FUNCTION_BLOCK FB_HomeNC_Test EXTENDS FB_TestSuite
VAR
    fbAxisRef : ARRAY [1..8] OF AXIS_REF;
    fbLimSwStatus : ARRAY [1..8] OF FB_LimSwStatus_TestDouble;
    //fbMotionLogger : FB_MotionLogger;
    fbMotionLogger : ARRAY [1..8] OF FB_MotionLogger;
    fbPower : ARRAY [1..8] OF FB_PowerNC[	(AxisRef := fbAxisRef[1]),
                                            (AxisRef := fbAxisRef[2]),
                                            (AxisRef := fbAxisRef[3]),
                                            (AxisRef := fbAxisRef[4]),
                                            (AxisRef := fbAxisRef[5]),
                                            (AxisRef := fbAxisRef[6]),
                                            (AxisRef := fbAxisRef[7]),
                                            (AxisRef := fbAxisRef[8])
                                            ];
END_VAR

GivenHomeCmdNoneThenHomeDoneIsTrue_Test1();
GivenHomeCmdAbsoluteSetThenThenAndHomeDoneAndPositionSetToUserDefineOffset_Test2();
GivenHomeCmdLowLimitModeAndABackwardSwPulseThenHomeDoneAndPositionSetToUserDefineOffset_Test3();
GivenHomeCmdSetToHighLimitAndHighLimitPulseThenHomeDoneAndPositionSetToUserDefineOffset_Test4();
GivenHomeCmdSetToHomeViaHighLimitAndHomeHighLimitPulseThenHomeDoneAndPositionSetToUserDefineOffset_Test5();
GivenHomeCmdSetToHomeViaLowLimitAndHomeLowLimitPulseThenHomeDoneAndPositionSetToUserDefineOffset_Test6();
GivenHomeCmdSetToHomeViaLowLimitAndBackwardLimitPulsebeforeHomeLowLimitIdexPulseThenHomeDoneAndPositionSetToUserDefineOffset_Test7();
GivenHomeCmdSetToHomeViaHighLimitAndForwardLimitPulsebeforeHomeHighLimitIdexPulseThenHomeDoneAndPositionSetToUserDefineOffset_Test8();

METHOD PRIVATE GivenHomeCmdAbsoluteSetThenThenAndHomeDoneAndPositionSetToUserDefineOffset_Test2
VAR_INST
    fbHome : FB_HomeNC(AxisRef:=fbAxisRef[2], iLimSwStatus:=fbLimSwStatus[2],iMotionLogger:=fbMotionLogger[2]):=(Mode:=E_EpicsHomeCmd.ABSOLUTE_SET);
    fbTestTimer: TON := (IN:=TRUE, PT:=T#8S);

    nTestStep : INT;
    fExpectedPosition : LREAL := 20.0;
    fActPosition : LREAL;
    bCalibrated : BOOL;
END_VAR
TEST(__POUNAME());

fbLimSwStatus[2]();
fbMotionLogger[2]();
// This methd must be called cyclicly
fbPower[2].Power(	Enable:=TRUE,
                     Enable_Positive:=fbLimSwStatus[2].LimForward,
                       Enable_Negative:=fbLimSwStatus[2].LimBackward,
                       Override:=100.0
                );

CASE nTestStep OF
    0:
        IF fbPower[2].PowerIsEnabled THEN
            fbHome.Home(Position:=20.0,BufferMode:=MC_BufferMode.MC_Aborting);
            nTestStep := nTestStep + 1;
        END_IF
    1:
        IF fbHome.Done THEN
            nTestStep := nTestStep + 1;
        END_IF
    2:
     //
END_CASE
fbAxisRef[2].ReadStatus();
fbHome();
fbTestTimer(IN := TRUE);

IF nTestStep = 2 THEN
bCalibrated := fbHome.Done;
AssertEquals_BOOL(Expected:=fbAxisRef[2].Status.Homed, Actual:=bCalibrated, Message := 'Axis not calibrated #1');

AssertEquals_LREAL ( Delta:=0.001, Expected:=fExpectedPosition, Actual:=fbAxisRef[2].NcToPlc.ActPos, Message:='Position is not the expected #2');
TEST_FINISHED();
ELSIF fbTestTimer.Q THEN
    AssertTrue(
        Condition := FALSE,
        Message := CONCAT('Timed out at step: ', TO_STRING(nTestStep))
    );
    TEST_FINISHED();
END_IF
END_METHOD

METHOD PRIVATE GivenHomeCmdLowLimitModeAndABackwardSwPulseThenHomeDoneAndPositionSetToUserDefineOffset_Test3
VAR_INST
    fbHome : FB_HomeNC(AxisRef:=fbAxisRef[3], iLimSwStatus:=fbLimSwStatus[3],iMotionLogger:=fbMotionLogger[3]):=(Mode:=E_EpicsHomeCmd.LOW_LIMIT);
    fbTestTimer: TON := (IN:=TRUE, PT:=T#5S);
    fbCamSwitchPulserSearch: TON := (IN:=TRUE, PT:=T#500MS);
    fbCamSwitchPulserSync: TON := (PT:=T#1000MS);
    nTestStep : INT;
    fExpectedPosition : LREAL := 20.0;
    fActPosition : LREAL;
    bCalibrated: BOOL;
    // reset this when error or homeDone
    bHomingOverride : BOOL := TRUE;
END_VAR
TEST(__POUNAME());

fbLimSwStatus[3]();
fbMotionLogger[3]();
fbPower[3].Power(	Enable:=TRUE,
                            Enable_Positive:=bHomingOverride OR fbLimSwStatus[3].LimForward,
                            Enable_Negative:=bHomingOverride OR fbLimSwStatus[3].LimBackward,
                            Override:=100.0);

CASE nTestStep OF
    0:
        IF fbPower[3].PowerIsEnabled THEN
            fbHome.Home(Position:=20.0,BufferMode:=MC_BufferMode.MC_Aborting);
            nTestStep := nTestStep + 1;
        END_IF

    1:
        IF fbCamSwitchPulserSearch.Q THEN
            fbLimSwStatus[3].LimBackward := FALSE;
            fbCamSwitchPulserSearch.IN := FALSE;
            fbCamSwitchPulserSync.IN := TRUE;
            nTestStep := nTestStep + 1;
        END_IF
    2:
        IF fbCamSwitchPulserSync.Q THEN
            fbLimSwStatus[3].LimBackward := TRUE;
            nTestStep := nTestStep + 1;
        END_IF
    3:
        IF fbHome.Done THEN
            nTestStep := nTestStep + 1;
        END_IF
    4:;
END_CASE
fbAxisRef[3].ReadStatus();
fbHome();
fbCamSwitchPulserSearch();
fbCamSwitchPulserSync();
fbTestTimer();

IF nTestStep = 4 THEN
    bCalibrated := fbHome.Done;
    AssertEquals_BOOL(Expected:=fbAxisRef[3].Status.Homed, Actual:=bCalibrated, Message := 'Axis not calibrated #1');
    AssertEquals_LREAL ( Delta:=0.001, Expected:=fExpectedPosition, Actual:=fbAxisRef[3].NcToPlc.ActPos, Message:='Position is not the expected #2');
    TEST_FINISHED();
ELSIF fbTestTimer.Q THEN
    AssertTrue(
        Condition := FALSE,
        Message := CONCAT('Timed out at step: ', TO_STRING(nTestStep))
    );

    TEST_FINISHED();
END_IF
END_METHOD

METHOD PRIVATE GivenHomeCmdNoneThenHomeDoneIsTrue_Test1
VAR_INST
    fbHome : FB_HomeNC(AxisRef:=fbAxisRef[1], iLimSwStatus:=fbLimSwStatus[1],iMotionLogger:=fbMotionLogger[1]):=(Mode:= E_EpicsHomeCmd.NONE);
    fbTestTimer: TON := (IN:=TRUE, PT:=T#5S);
    nTestStep : INT;
END_VAR
TEST(__POUNAME());

fbLimSwStatus[1]();
fbMotionLogger[1]();

CASE nTestStep OF
    0:

        fbPower[1].Power(	Enable:=TRUE,
                            Enable_Positive:=fbLimSwStatus[1].LimForward,
                            Enable_Negative:=fbLimSwStatus[1].LimBackward,
                            Override:=100.0);
        nTestStep := nTestStep + 1;
    1:
    IF fbPower[1].PowerIsEnabled THEN
        fbHome.Home(Position:=0.0,BufferMode:=MC_BufferMode.MC_Aborting);
        nTestStep := nTestStep + 1;
    END_IF

    2:
        IF fbHome.Done THEN
            nTestStep := nTestStep + 1;
        END_IF
    3:
     //
END_CASE

fbPower[1]();
fbHome();

fbTestTimer(IN := TRUE);

IF nTestStep = 3 THEN

    TEST_FINISHED();
ELSIF fbTestTimer.Q THEN
    AssertTrue(
        Condition := FALSE,
        Message := CONCAT('Timed out at step: ', TO_STRING(nTestStep))
    );

    TEST_FINISHED();
END_IF
END_METHOD

METHOD PRIVATE GivenHomeCmdSetToHighLimitAndHighLimitPulseThenHomeDoneAndPositionSetToUserDefineOffset_Test4
VAR_INST
    fbHome : FB_HomeNC(AxisRef:=fbAxisRef[4], iLimSwStatus:=fbLimSwStatus[4],iMotionLogger:=fbMotionLogger[4]):=(Mode:=E_EpicsHomeCmd.HIGH_LIMIT);
    fbTestTimer: TON := (IN:=TRUE, PT:=T#5S);
    fbCamSwitchPulserSearch: TON := (IN:=TRUE, PT:=T#500MS);
    fbCamSwitchPulserSync: TON := (PT:=T#1000MS);
    nTestStep : INT;
    fExpectedPosition : LREAL := 20.0;
    fActPosition : LREAL;
    bCalibrated: BOOL;
    // reset this when error or homeDone
    bHomingOverride : BOOL := TRUE;
END_VAR
TEST(__POUNAME());

fbLimSwStatus[4]();
fbMotionLogger[4]();
fbPower[4].Power(	Enable:=TRUE,
                            Enable_Positive:=bHomingOverride OR fbLimSwStatus[4].LimForward,
                            Enable_Negative:=bHomingOverride OR fbLimSwStatus[4].LimBackward,
                            Override:=100.0);

CASE nTestStep OF
    0:
        IF fbPower[4].PowerIsEnabled THEN
            fbHome.Home(Position:=20.0,BufferMode:=MC_BufferMode.MC_Aborting);
            nTestStep := nTestStep + 1;
        END_IF

    1:
        IF fbCamSwitchPulserSearch.Q THEN
            fbLimSwStatus[4].LimForward := FALSE;
            fbCamSwitchPulserSearch.IN := FALSE;
            fbCamSwitchPulserSync.IN := TRUE;
            nTestStep := nTestStep + 1;
        END_IF
    2:
        IF fbCamSwitchPulserSync.Q THEN
            fbLimSwStatus[4].LimForward := TRUE;
            nTestStep := nTestStep + 1;
        END_IF
    3:
        IF fbHome.Done THEN
            nTestStep := nTestStep + 1;
        END_IF
    4:;
END_CASE
fbAxisRef[4].ReadStatus();
fbHome();
fbCamSwitchPulserSearch();
fbCamSwitchPulserSync();
fbTestTimer();

IF nTestStep = 4 THEN
    bCalibrated := fbHome.Done;
    AssertEquals_BOOL(Expected:=fbAxisRef[4].Status.Homed, Actual:=bCalibrated, Message := 'Axis not calibrated #1');
    AssertEquals_LREAL ( Delta:=0.001, Expected:=fExpectedPosition, Actual:=fbAxisRef[4].NcToPlc.ActPos, Message:='Position is not the expected #2');
    TEST_FINISHED();
ELSIF fbTestTimer.Q THEN
    AssertTrue(
        Condition := FALSE,
        Message := CONCAT('Timed out at step: ', TO_STRING(nTestStep))
    );

    TEST_FINISHED();
END_IF
END_METHOD

METHOD PRIVATE GivenHomeCmdSetToHomeViaHighLimitAndForwardLimitPulsebeforeHomeHighLimitIdexPulseThenHomeDoneAndPositionSetToUserDefineOffset_Test8
VAR_INST
    fbHome : FB_HomeNC(AxisRef:=fbAxisRef[8], iLimSwStatus:=fbLimSwStatus[8],iMotionLogger:=fbMotionLogger[8]):=(Mode:= E_EpicsHomeCmd.HOME_VIA_HIGH);
    fbTestTimer: TON := (IN:=TRUE, PT:=T#5S);
    fbCamSwitchPulserSearch: TON := (IN:=TRUE, PT:=T#500MS);
    fbCamSwitchPulserSync: TON := (PT:=T#1000MS);
    nTestStep : INT;
    fExpectedPosition : LREAL := 20.0;
    fActPosition : LREAL;
    bCalibrated: BOOL;
    // reset this when error or homeDone
    bHomingOverride : BOOL := TRUE;

END_VAR
TEST(__POUNAME());
fbAxisRef[8].ReadStatus();
fbLimSwStatus[8]();
fbMotionLogger[8]();
fbPower[8].Power(	Enable:=TRUE,
                            Enable_Positive:=bHomingOverride OR fbLimSwStatus[8].LimForward,
                            Enable_Negative:=bHomingOverride OR fbLimSwStatus[8].LimForward,
                            Override:=100.0);
CASE nTestStep OF
    0:
        IF fbPower[8].PowerIsEnabled THEN
            fbHome.Home(Position:=20.0,BufferMode:=MC_BufferMode.MC_Aborting);
            nTestStep := nTestStep + 1;
        END_IF
    1:
        IF fbCamSwitchPulserSearch.Q THEN
            fbLimSwStatus[8].LimForward := FALSE;
            fbCamSwitchPulserSearch.IN := FALSE;
            fbCamSwitchPulserSync.IN := TRUE;
            nTestStep := nTestStep + 1;
        END_IF
    2:
        IF fbCamSwitchPulserSync.Q THEN
            fbLimSwStatus[8].LimForward := TRUE;
            nTestStep := nTestStep + 1;
        END_IF
    3:
        IF fbHome.HLDone THEN
            // prepare second stage homing
            fbCamSwitchPulserSearch.IN := TRUE;
            fbCamSwitchPulserSync.IN := FALSE;
            nTestStep := nTestStep + 1;
        END_IF
    4:
        IF fbCamSwitchPulserSearch.Q THEN
            fbLimSwStatus[8].LimHome := TRUE;
            fbCamSwitchPulserSearch.IN := FALSE;
            fbCamSwitchPulserSync.IN := TRUE;
            nTestStep := nTestStep + 1;
        END_IF
    5:
        IF fbCamSwitchPulserSync.Q THEN
            fbLimSwStatus[8].LimHome := FALSE;
            nTestStep := nTestStep + 1;
        END_IF
    6:
        IF fbHome.Done THEN
            nTestStep := nTestStep + 1;
        END_IF
    7:;
END_CASE

fbPower[8]();
fbHome();

fbCamSwitchPulserSearch();
fbCamSwitchPulserSync();
fbTestTimer();

IF nTestStep = 7 THEN
    bCalibrated := fbHome.Done;
    AssertEquals_BOOL(Expected:=fbAxisRef[8].Status.Homed, Actual:=bCalibrated, Message := 'Axis not calibrated #1');
    AssertEquals_LREAL ( Delta:=0.001, Expected:=fExpectedPosition, Actual:=fbAxisRef[8].NcToPlc.ActPos, Message:='Position is not the expected #2');
    TEST_FINISHED();
ELSIF fbTestTimer.Q THEN
    AssertTrue(
        Condition := FALSE,
        Message := CONCAT('Timed out at step: ', TO_STRING(nTestStep))
    );

    TEST_FINISHED();
END_IF
END_METHOD

METHOD PRIVATE GivenHomeCmdSetToHomeViaHighLimitAndHomeHighLimitPulseThenHomeDoneAndPositionSetToUserDefineOffset_Test5
VAR_INST
    fbHome : FB_HomeNC(AxisRef:=fbAxisRef[5], iLimSwStatus:=fbLimSwStatus[5],iMotionLogger:=fbMotionLogger[5]):=(Mode:= E_EpicsHomeCmd.HOME_VIA_HIGH);
    fbTestTimer: TON := (IN:=TRUE, PT:=T#5S);
    fbCamSwitchPulserSearch: TON := (IN:=TRUE, PT:=T#500MS);
    fbCamSwitchPulserSync: TON := (PT:=T#1000MS);
    nTestStep : INT;
    fExpectedPosition : LREAL := 20.0;
    fActPosition : LREAL;
    bCalibrated: BOOL;
    // reset this when error or homeDone
    bHomingOverride : BOOL := TRUE;

END_VAR
TEST(__POUNAME());

fbLimSwStatus[5]();
fbMotionLogger[5]();
fbPower[5].Power(	Enable:=TRUE,
                            Enable_Positive:=bHomingOverride OR fbLimSwStatus[5].LimForward,
                            Enable_Negative:=bHomingOverride OR fbLimSwStatus[5].LimBackward,
                            Override:=100.0);
CASE nTestStep OF
    0:
        IF fbPower[5].PowerIsEnabled THEN
            fbHome.Home(Position:=20.0,BufferMode:=MC_BufferMode.MC_Aborting);
            nTestStep := nTestStep + 1;
        END_IF
    1:
        IF fbCamSwitchPulserSearch.Q THEN
            fbLimSwStatus[5].LimHome := TRUE;
            fbCamSwitchPulserSearch.IN := FALSE;
            fbCamSwitchPulserSync.IN := TRUE;
            nTestStep := nTestStep + 1;
        END_IF
    2:
        IF fbCamSwitchPulserSync.Q THEN
            fbLimSwStatus[5].LimHome := FALSE;
            nTestStep := nTestStep + 1;
        END_IF
    3:
        IF fbHome.Done THEN
            nTestStep := nTestStep + 1;
        END_IF
    4:;
END_CASE
fbAxisRef[5].ReadStatus();
fbPower[5]();
fbHome();

fbCamSwitchPulserSearch();
fbCamSwitchPulserSync();
fbTestTimer();

IF nTestStep = 4 THEN
    bCalibrated := fbHome.Done;
    AssertEquals_BOOL(Expected:=fbAxisRef[5].Status.Homed, Actual:=bCalibrated, Message := 'Axis not calibrated #1');
    AssertEquals_LREAL ( Delta:=0.001, Expected:=fExpectedPosition, Actual:=fbAxisRef[5].NcToPlc.ActPos, Message:='Position is not the expected #2');
    TEST_FINISHED();
ELSIF fbTestTimer.Q THEN
    AssertTrue(
        Condition := FALSE,
        Message := CONCAT('Timed out at step: ', TO_STRING(nTestStep))
    );

    TEST_FINISHED();
END_IF
END_METHOD

METHOD PRIVATE GivenHomeCmdSetToHomeViaLowLimitAndBackwardLimitPulsebeforeHomeLowLimitIdexPulseThenHomeDoneAndPositionSetToUserDefineOffset_Test7
VAR_INST
    fbHome : FB_HomeNC(AxisRef:=fbAxisRef[7], iLimSwStatus:=fbLimSwStatus[7],iMotionLogger:=fbMotionLogger[7]):=(Mode:= E_EpicsHomeCmd.HOME_VIA_LOW);
    fbTestTimer: TON := (IN:=TRUE, PT:=T#5S);
    fbCamSwitchPulserSearch: TON := (IN:=TRUE, PT:=T#500MS);
    fbCamSwitchPulserSync: TON := (PT:=T#1000MS);
    nTestStep : INT;
    fExpectedPosition : LREAL := 20.0;
    fActPosition : LREAL;
        bCalibrated: BOOL;
    // reset this when error or homeDone
    bHomingOverride : BOOL := TRUE;

END_VAR
TEST(__POUNAME());
fbAxisRef[7].ReadStatus();
fbLimSwStatus[7]();
fbMotionLogger[7]();
fbPower[7].Power(	Enable:=TRUE,
                            Enable_Positive:=bHomingOverride OR fbLimSwStatus[7].LimForward,
                            Enable_Negative:=bHomingOverride OR fbLimSwStatus[7].LimBackward,
                            Override:=100.0);
CASE nTestStep OF
    0:
        IF fbPower[7].PowerIsEnabled THEN
            fbHome.Home(Position:=20.0,BufferMode:=MC_BufferMode.MC_Aborting);
            nTestStep := nTestStep + 1;
        END_IF
    1:
        IF fbCamSwitchPulserSearch.Q THEN
            fbLimSwStatus[7].LimBackward := FALSE;
            fbCamSwitchPulserSearch.IN := FALSE;
            fbCamSwitchPulserSync.IN := TRUE;
            nTestStep := nTestStep + 1;
        END_IF
    2:
        IF fbCamSwitchPulserSync.Q THEN
            fbLimSwStatus[7].LimBackward := TRUE;
            nTestStep := nTestStep + 1;
        END_IF
    3:
        IF fbHome.HLDone THEN
            // prepare second stage homing
            fbCamSwitchPulserSearch.IN := TRUE;
            fbCamSwitchPulserSync.IN := FALSE;
            nTestStep := nTestStep + 1;
        END_IF
    4:
        IF fbCamSwitchPulserSearch.Q THEN
            fbLimSwStatus[7].LimHome := TRUE;
            fbCamSwitchPulserSearch.IN := FALSE;
            fbCamSwitchPulserSync.IN := TRUE;
            nTestStep := nTestStep + 1;
        END_IF
    5:
        IF fbCamSwitchPulserSync.Q THEN
            fbLimSwStatus[7].LimHome := FALSE;
            nTestStep := nTestStep + 1;
        END_IF
    6:
        IF fbHome.Done THEN
            nTestStep := nTestStep + 1;
        END_IF
    7:;
END_CASE

fbPower[7]();
fbHome();

fbCamSwitchPulserSearch();
fbCamSwitchPulserSync();
fbTestTimer();

IF nTestStep = 7 THEN
    bCalibrated := fbHome.Done;
    AssertEquals_BOOL(Expected:=fbAxisRef[7].Status.Homed, Actual:=bCalibrated, Message := 'Axis not calibrated #1');
    AssertEquals_LREAL ( Delta:=0.001, Expected:=fExpectedPosition, Actual:=fbAxisRef[7].NcToPlc.ActPos, Message:='Position is not the expected #2');
    TEST_FINISHED();
ELSIF fbTestTimer.Q THEN
    AssertTrue(
        Condition := FALSE,
        Message := CONCAT('Timed out at step: ', TO_STRING(nTestStep))
    );

    TEST_FINISHED();
END_IF
END_METHOD

METHOD PRIVATE GivenHomeCmdSetToHomeViaLowLimitAndHomeLowLimitPulseThenHomeDoneAndPositionSetToUserDefineOffset_Test6
VAR_INST
    fbHome : FB_HomeNC(AxisRef:=fbAxisRef[6], iLimSwStatus:=fbLimSwStatus[6],iMotionLogger:=fbMotionLogger[6]):=(Mode:= E_EpicsHomeCmd.HOME_VIA_LOW);
    fbTestTimer: TON := (IN:=TRUE, PT:=T#5S);
    fbCamSwitchPulserSearch: TON := (IN:=TRUE, PT:=T#500MS);
    fbCamSwitchPulserSync: TON := (PT:=T#1000MS);
    nTestStep : INT;
    fExpectedPosition : LREAL := 20.0;
    fActPosition : LREAL;
        bCalibrated: BOOL;
    // reset this when error or homeDone
    bHomingOverride : BOOL := TRUE;

END_VAR
TEST(__POUNAME());

fbLimSwStatus[6]();
fbMotionLogger[6]();
fbPower[6].Power(	Enable:=TRUE,
                            Enable_Positive:=bHomingOverride OR fbLimSwStatus[6].LimForward,
                            Enable_Negative:=bHomingOverride OR fbLimSwStatus[6].LimBackward,
                            Override:=100.0);
CASE nTestStep OF
    0:
        IF fbPower[6].PowerIsEnabled THEN
            fbHome.Home(Position:=20.0,BufferMode:=MC_BufferMode.MC_Aborting);
            nTestStep := nTestStep + 1;
        END_IF
    1:
        IF fbCamSwitchPulserSearch.Q THEN
            fbLimSwStatus[6].LimHome := TRUE;
            fbCamSwitchPulserSearch.IN := FALSE;
            fbCamSwitchPulserSync.IN := TRUE;
            nTestStep := nTestStep + 1;
        END_IF
    2:
        IF fbCamSwitchPulserSync.Q THEN
            fbLimSwStatus[6].LimHome := FALSE;
            nTestStep := nTestStep + 1;
        END_IF
    3:
        IF fbHome.Done THEN
            nTestStep := nTestStep + 1;
        END_IF
    4:;
END_CASE
fbAxisRef[6].ReadStatus();
fbPower[6]();
fbHome();

fbCamSwitchPulserSearch();
fbCamSwitchPulserSync();
fbTestTimer();

IF nTestStep = 4 THEN
    bCalibrated := fbHome.Done;
    AssertEquals_BOOL(Expected:=fbAxisRef[6].Status.Homed, Actual:=bCalibrated, Message := 'Axis not calibrated #1');
    AssertEquals_LREAL ( Delta:=0.001, Expected:=fExpectedPosition, Actual:=fbAxisRef[6].NcToPlc.ActPos, Message:='Position is not the expected #2');
    TEST_FINISHED();
ELSIF fbTestTimer.Q THEN
    AssertTrue(
        Condition := FALSE,
        Message := CONCAT('Timed out at step: ', TO_STRING(nTestStep))
    );

    TEST_FINISHED();
END_IF
END_METHOD

END_FUNCTION_BLOCK

(* stored: Version 1.1.0.1
   POU FB_HomeNC_Test: Id {0f089b23-a654-4e4f-b104-c56af0e6d9b3}, SpecialFunc None
   Method GivenHomeCmdAbsoluteSetThenThenAndHomeDoneAndPositionSetToUserDefineOffset_Test2: Id {d4754e57-693c-40b7-9460-2ffc5ab4a21b}
   Method GivenHomeCmdLowLimitModeAndABackwardSwPulseThenHomeDoneAndPositionSetToUserDefineOffset_Test3: Id {258c5fca-fb29-4806-85ec-0c0567cfff16}
   Method GivenHomeCmdNoneThenHomeDoneIsTrue_Test1: Id {828068d5-3f4b-4e81-8832-2d3b09781313}
   Method GivenHomeCmdSetToHighLimitAndHighLimitPulseThenHomeDoneAndPositionSetToUserDefineOffset_Test4: Id {d6dfc9cc-8559-4032-bc50-ad12f2b74624}
   Method GivenHomeCmdSetToHomeViaHighLimitAndForwardLimitPulsebeforeHomeHighLimitIdexPulseThenHomeDoneAndPositionSetToUserDefineOffset_Test8: Id {504926c1-1919-481e-bdb9-25f2e0554127}
   Method GivenHomeCmdSetToHomeViaHighLimitAndHomeHighLimitPulseThenHomeDoneAndPositionSetToUserDefineOffset_Test5: Id {b2085644-7959-47fa-a9ee-a37dd04f378f}
   Method GivenHomeCmdSetToHomeViaLowLimitAndBackwardLimitPulsebeforeHomeLowLimitIdexPulseThenHomeDoneAndPositionSetToUserDefineOffset_Test7: Id {ce7122bb-2e16-4f97-b955-1e752383c80f}
   Method GivenHomeCmdSetToHomeViaLowLimitAndHomeLowLimitPulseThenHomeDoneAndPositionSetToUserDefineOffset_Test6: Id {40dcb32c-5f70-434b-a8dd-25a5277ca8f8} *)
